// SIMATIC S7-200 SMART project (STEP 7-Micro/WIN SMART), CPU SR40

SYMBOL_TABLE 系统符号
First_Scan_On    SM0.1    // 仅在第一个扫描周期时接通
END_SYMBOL_TABLE

ORGANIZATION_BLOCK MAIN:OB1
TITLE=程序注释
BEGIN
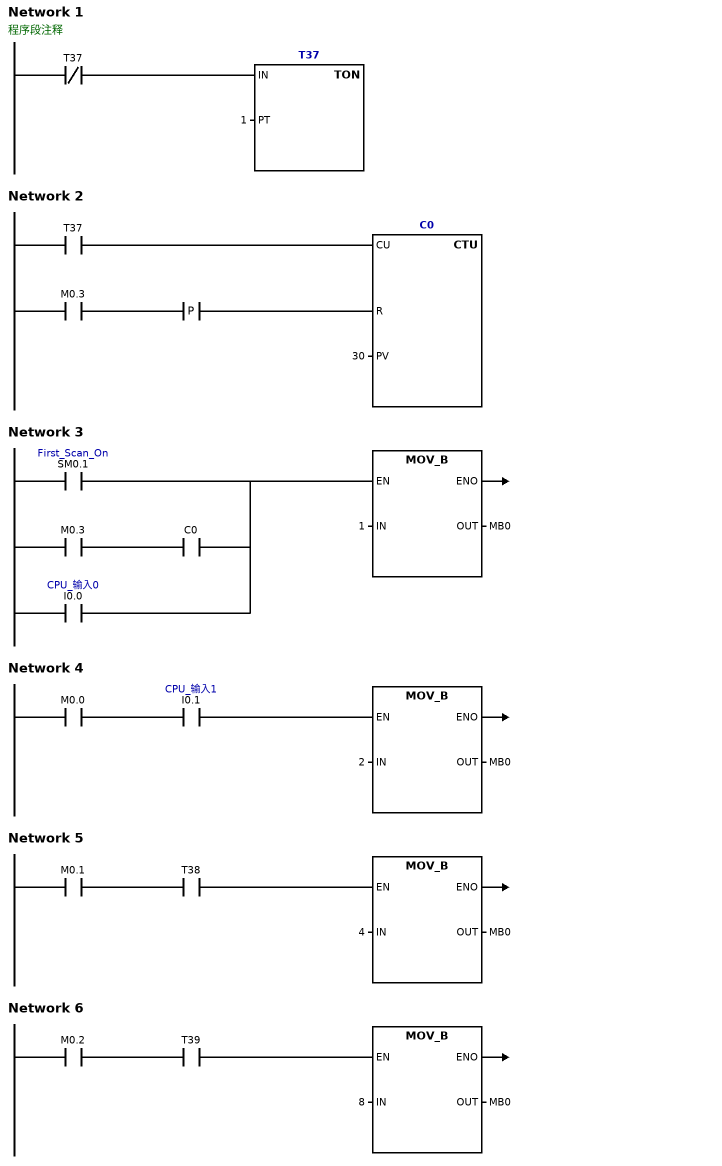
Network 1
// 程序段注释
LDN    T37
TON    T37, 1
Network 2
LD     T37
LD     M0.3
EU
CTU    C0, 30
Network 3
LD     First_Scan_On:SM0.1
LD     M0.3
A      C0
OLD
O      CPU_输入0:I0.0
MOVB   1, MB0
Network 4
LD     M0.0
A      CPU_输入1:I0.1
MOVB   2, MB0
Network 5
LD     M0.1
A      T38
MOVB   4, MB0
Network 6
LD     M0.2
A      T39
MOVB   8, MB0
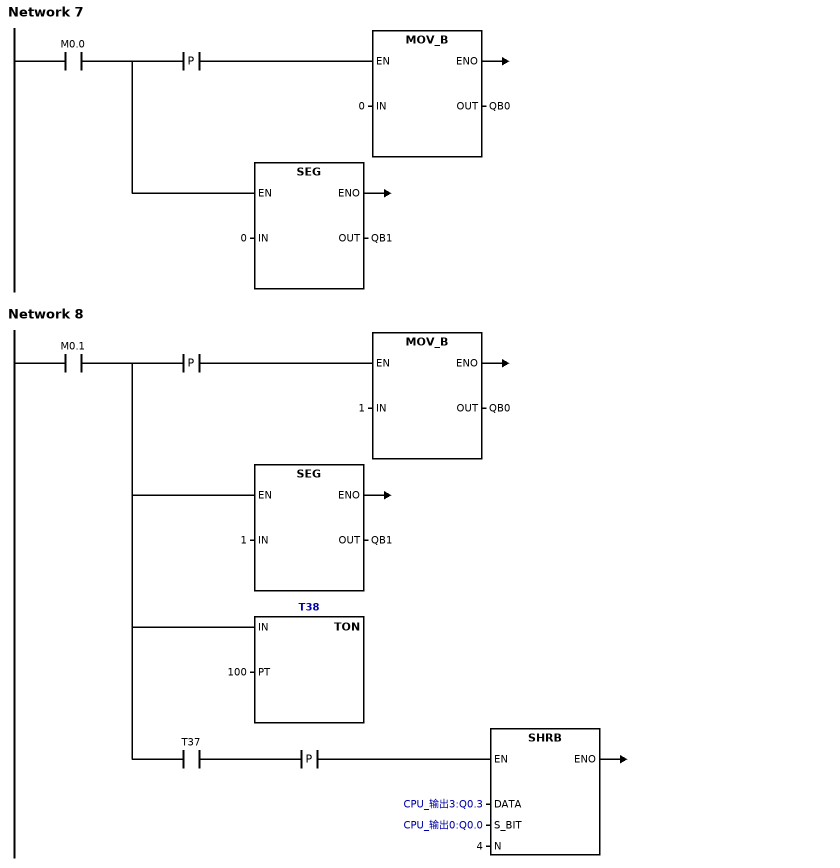
Network 7
LD     M0.0
LPS
EU
MOVB   0, QB0
LPP
SEG    0, QB1
Network 8
LD     M0.1
LPS
EU
MOVB   1, QB0
LRD
SEG    1, QB1
LRD
TON    T38, 100
LPP
A      T37
EU
SHRB   CPU_输出3:Q0.3, CPU_输出0:Q0.0, 4
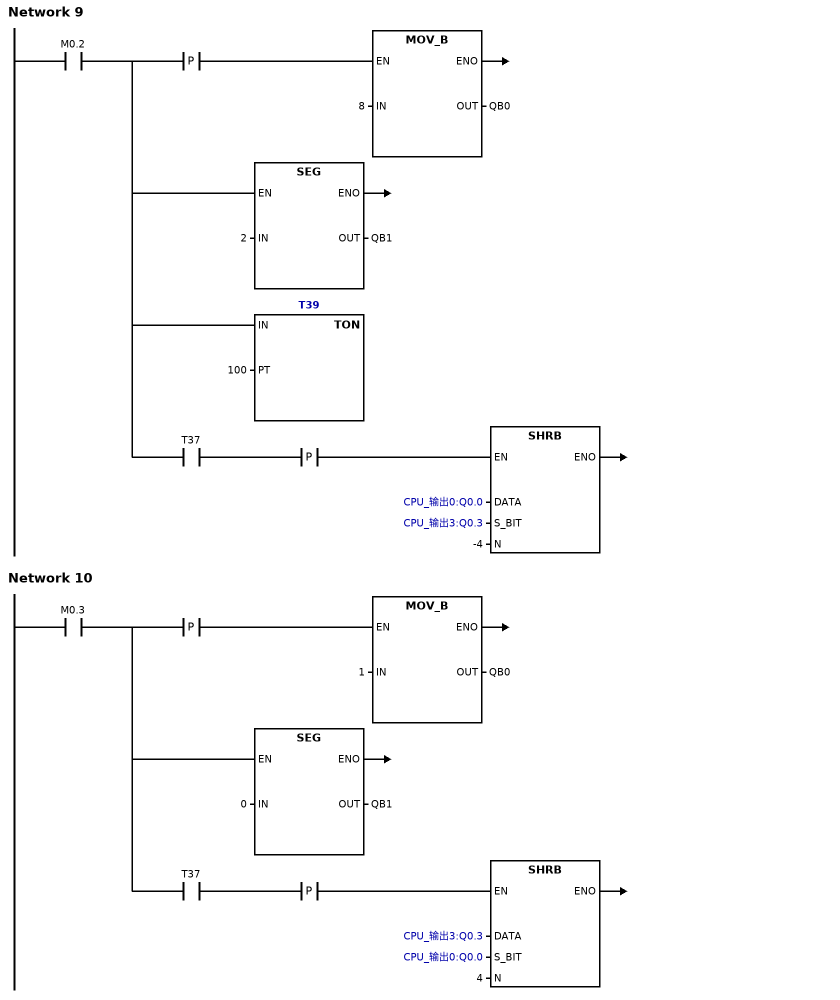
Network 9
LD     M0.2
LPS
EU
MOVB   8, QB0
LRD
SEG    2, QB1
LRD
TON    T39, 100
LPP
A      T37
EU
SHRB   CPU_输出0:Q0.0, CPU_输出3:Q0.3, -4
Network 10
LD     M0.3
LPS
EU
MOVB   1, QB0
LRD
SEG    0, QB1
LPP
A      T37
EU
SHRB   CPU_输出3:Q0.3, CPU_输出0:Q0.0, 4
END_ORGANIZATION_BLOCK
